FUNCTION_BLOCK Base
VAR_INPUT
END_VAR
VAR_OUTPUT
END_VAR
VAR
END_VAR

END_FUNCTION_BLOCK

(* stored: Version 1.1.0.1
   POU Base: Id {f1f9ec23-3003-4cf0-ab47-c55ac500b671}, SpecialFunc None *)
